FUNCTION_BLOCK JackGripper
  (* Standard: 61499-2 *)
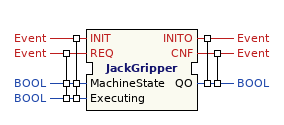
  EVENT_INPUT
    INIT WITH MachineState, Executing;
    REQ WITH MachineState, Executing;
  END_EVENT
  EVENT_OUTPUT
    INITO WITH QO;
    CNF WITH QO;
  END_EVENT
  VAR_INPUT
    MachineState : BOOL;
    Executing : BOOL;
  END_VAR
  VAR_OUTPUT
    QO : BOOL;
  END_VAR
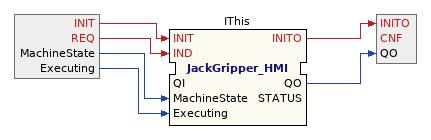
  FBS
    IThis : JackGripper_HMI;
  END_FBS
  EVENT_CONNECTIONS
    INIT TO IThis.INIT;
    REQ TO IThis.IND;
    IThis.INITO TO INITO;
  END_CONNECTIONS
  DATA_CONNECTIONS
    MachineState TO IThis.MachineState;
    Executing TO IThis.Executing;
    IThis.QO TO QO;
  END_CONNECTIONS
END_FUNCTION_BLOCK
